# EPICS autosave request: ADApp/Db/NDFileNetCDF_settings.req
file "NDPluginFile_settings.req", P=$(P), R=$(R)
